FUNCTION_BLOCK FB_Robot EXTENDS FB_EquipmentModule_SR
VAR
    // Sub module definitions here

    // List of sub modules

    ipSubModules_Init : ARRAY[1..Parameters_PackML_Base.MAX_NO_OF_SUBMODULES] OF I_PackML_BaseModule := [];

    // Component definitions here

    Robot : FB_Component_Robot := (Name := 'Robot');

END_VAR

VAR

    //Properties
    DetailIndex : UDINT := 1;

    Handshake_Step : DINT;

    _DryRun : BOOL;

END_VAR

METHOD PROTECTED Aborting
VAR_INPUT
END_VAR
Handshake_Step                      := 0;
Robot.Handshake.OUT.Execute_Step    := FALSE;
Robot.Handshake.OUT.Execute_StepNum := 0;
DetailIndex                         := 1;

Super^.Aborting();
END_METHOD

METHOD PROTECTED Clearing
VAR_INPUT
END_VAR
Super^.Clearing();
END_METHOD

METHOD PROTECTED Completing
VAR_INPUT
END_VAR
Super^.Completing();
END_METHOD

METHOD CyclicLogic
VAR_INPUT
END_VAR

VAR

END_VAR
IF NOT _InitComplete THEN
    _InitComplete := Initialize();
    RETURN;
END_IF

//SimulationOn();

// transfer var from EM to COMP

// IF _Name = 'Robot 1' THEN

//     Robot.RobotType := 'Handling';

// ELSIF _Name = 'Robot 2' OR _Name = 'Robot 3' THEN

//     Robot.RobotType := 'Fastening';

// END_IF

SUPER^.CyclicLogic();
END_METHOD

METHOD CyclicLogicSimulation : BOOL
VAR_INPUT
END_VAR
END_METHOD

PROPERTY DryRun : BOOL
GET
DryRun := _DryRun;
END_GET
SET
_DryRun := DryRun;
END_SET
END_PROPERTY

METHOD PROTECTED Execute
VAR_INPUT
END_VAR
//  logic
WaitSync_Robot();

SubModuleMonitor();

SUPER^.Execute();
END_METHOD

METHOD ExtractNumFromString : DINT
VAR_INPUT
    InputString : STRING;
END_VAR

VAR
    NumberString : STRING     := ''; // Temporary string to collect digits
    Numbers      : STRING[10] := '0123456789'; // Temporary string to collect digits
    CurrentChar  : BYTE; // Current character being processed
    Result       : UDINT := 0; // Final extracted number as UDINT
    i            : INT   := 1; // String index
END_VAR
ExtractNumFromString := 0;
j                    := 0;

FOR i := 0 TO LEN(InputString) DO
    CurrentChar := InputString[i];

    // Check if the current character is a digit
    IF CurrentChar >= Numbers[0] AND CurrentChar <= Numbers[9] THEN
        NumberString[j] := CurrentChar;
        j               := j + 1;
    END_IF
END_FOR

// Check for a number at the end of the string
IF LEN(NumberString) > 0 THEN
    ExtractNumFromString := STRING_TO_DINT(NumberString); // Convert to UDINT
END_IF
END_METHOD

METHOD HMIControl
VAR_INPUT
END_VAR
END_METHOD

METHOD PROTECTED Holding
VAR_INPUT
END_VAR
IF Robot.Handshake.IN.TaskRunning = FALSE THEN
    SUPER^.Holding();
END_IF
END_METHOD

//! @summary Basic module initialization logic
METHOD PROTECTED Initialize : BOOL;
VAR
    i                        : UDINT;
    varInfo                  : __SYSTEM.VAR_INFO;
    AllSubUnitsInitialized   : BOOL := TRUE;
    AllComponentsInitialized : BOOL := TRUE;
END_VAR

//! @description This method is called by <c>CyclicLogic()</c> as required
Initialize := FALSE;

CASE DescendantSequenceState OF
    0:
        RegisterComponent(Robot);

        _LogModeChanges         := FALSE;
        _LogStateChanges        := FALSE;
        DescendantSequenceState := DescendantSequenceState + 10;

    10:
        //Setup Custom modes here

        (*CustomModes(eMode                          :=,
                    sName                          :=,
                    bDisableClearing               :=,
                    bDisableStarting               :=,
                    bDisableSuspended              :=,
                    bDisableStopping               :=,
                    bDisableAborting               :=,
                    bDisableHolding                :=,
                    bDisableHeld                   :=,
                    bDisableUnholding              :=,
                    bDisableSuspending             :=,
                    bDisableUnsuspending           :=,
                    bDisableResetting              :=,
                    bDisableIdle                   :=,
                    bDisableCompleting             :=,
                    bDisableComplete               :=,
                    bEnableUnitModeChangeStopped   :=,
                    bEnableUnitModeChangeIdle      :=,
                    bEnableUnitModeChangeSuspended :=,
                    bEnableUnitModeChangeExecute   :=,
                    bEnableUnitModeChangeAborted   :=,
                    bEnableUnitModeChangeHeld      :=,
                    bEnableUnitModeChangeComplete  :=,
                    bError                         =>,
                    nErrorId                       =>);*)

        DescendantSequenceState := DescendantSequenceState + 10;

    20:
        //Copy Mode names

        FOR i := 1 TO 3 DO
            ModeNames[i] := F_UnitModeToString(UDINT_TO_DINT(i));
        END_FOR

        RegisterExternalController(Controller := fbControlSourceHMI);
        fbControlSourceHMI.CyclicLogic();
        DescendantSequenceState := DescendantSequenceState + 10;

    30:
        //Call the Super

        IF SUPER^.Initialize() THEN
            DescendantSequenceState := DescendantSequenceState + 10;
        END_IF

    40:
        Initialize := TRUE;
END_CASE
END_METHOD

METHOD NailPlate : BOOL
VAR_INPUT
    Step : ST_CSV_Step;
END_VAR
// clear out array first
Robot.Clear_DataToSend();

// first entry is always step type
Robot.RecipeData_ToSend[1] := DINT_TO_USINT(E_CommandName.NailPlate);

// Robot.RecipeData_ToSend[2] := INT_TO_USINT(Plates[1].PlateNumber);
// 
// Robot.RecipeData_ToSend[3] := STRING_TO_USINT(Plates[1].PlateGauge);
// 
// Robot.RecipeData_ToSend[4] := LREAL_TO_USINT(TRUNC(Plates[1].PlateWidth * 10));
// 
// Robot.RecipeData_ToSend[5] := LREAL_TO_USINT(TRUNC(Plates[1].PlateHeight * 10));
// 
// Robot.RecipeData_ToSend[6] := LREAL_TO_USINT(TRUNC(Plates[1].PlatePlaceX * 10));
// 
// Robot.RecipeData_ToSend[7] := LREAL_TO_USINT(TRUNC(Plates[1].PlatePlaceY * 10));
// 
// Robot.RecipeData_ToSend[8] := LREAL_TO_USINT(TRUNC(Plates[1].PlatePlaceAngle * 10));
END_METHOD

PROPERTY OtherInputs : ARRAY[0..7] OF USINT
GET
OtherInputs := Robot.OtherInputs;
END_GET
END_PROPERTY

PROPERTY OtherOutputs : ARRAY[0..7] OF USINT
SET
Robot.OtherOutputs := OtherOutputs;
END_SET
END_PROPERTY

METHOD PROTECTED Resetting
VAR_INPUT
END_VAR
// reset handshake step
Handshake_Step                      := 0;
Robot.Handshake.OUT.Execute_Step    := FALSE;
Robot.Handshake.OUT.Execute_StepNum := 0;
DetailIndex                         := 1;

Super^.Resetting();
END_METHOD

METHOD PROTECTED Starting
VAR_INPUT
END_VAR
Handshake_Step                      := 0;
Robot.Handshake.OUT.Execute_Step    := FALSE;
Robot.Handshake.OUT.Execute_StepNum := 0;
DetailIndex                         := 1;

Super^.Starting();
END_METHOD

METHOD PROTECTED Stopping
VAR_INPUT
END_VAR
Super^.Stopping();
END_METHOD

(*! @summary This method monitors <b>submodules</b> within this PackML module and initiates fault responses as required*)
METHOD PROTECTED SubModuleMonitor : BOOL
SUPER^.SubModuleMonitor();
END_METHOD

METHOD PROTECTED Suspending
VAR_INPUT
END_VAR
IF Robot.Handshake.IN.TaskRunning = FALSE THEN
    SUPER^.Suspending();
END_IF
END_METHOD

METHOD PROTECTED Unholding
VAR_INPUT
END_VAR
SUPER^.Unholding();
END_METHOD

METHOD PROTECTED Unsuspending
VAR_INPUT
END_VAR
IF Robot.Handshake.IN.TaskRunning OR _InSimulation OR _ForceHold THEN
    SUPER^.Unsuspending();
END_IF
END_METHOD

METHOD WaitSync_Robot : BOOL
VAR
END_VAR

VAR_INST
    State : UDINT;
END_VAR
CASE State OF
    0:
        IF Robot.Handshake.IN.SubStepNumber > E_WaitSync.EMPTY THEN
            State := 1;
        END_IF

    1:
        _RequestedWaitSync := Robot.Handshake.IN.SubStepNumber;

        IF _RequestedWaitSync = _ResponseWaitSync THEN
            State := 2;
        END_IF

    2:
        Robot.Handshake.OUT.SubStepResponse := _ResponseWaitSync;

        IF Robot.Handshake.IN.SubStepNumber = E_WaitSync.EMPTY THEN
            _RequestedWaitSync := Robot.Handshake.IN.SubStepNumber;

            IF _ResponseWaitSync = E_WaitSync.EMPTY THEN
                Robot.Handshake.OUT.SubStepResponse := E_WaitSync.EMPTY;
                State                               := 0;
            END_IF
        END_IF

END_CASE
END_METHOD

END_FUNCTION_BLOCK

(* stored: Version 1.1.0.1
   POU FB_Robot: Id {1600db56-8704-42a5-b4ed-9569364dccae}, SpecialFunc None
   Folder I_CyclicFB: Id {f5633602-59b7-4bc0-9d4d-ad1c9ac3c89c}
   Folder Methods: Id {3c285524-643a-4343-a43c-a6df2c090b43}
   Folder ActingStates: Id {e4c87074-4e3f-4b79-aa36-c3b0b3bf226d}
   Folder CommandSteps: Id {61add708-9f29-4d83-adda-d2dcfb977e3f}
   Folder WaitingStates: Id {07ea4080-d9c0-4b39-9c64-a0a78873d1a8}
   Folder Properties: Id {e67c342a-5979-4627-bde3-a6f0dcd900b1}
   Method Aborting: Id {52fe1441-b0c0-423d-9d7a-ac2b065483cc}
   Method Clearing: Id {f68b84fa-c8c7-4a58-bb40-a12a77c808f3}
   Method Completing: Id {2b2dd47a-19b1-4d47-9ce0-79bec958c7ba}
   Method CyclicLogic: Id {86d8ffcb-cac6-4160-a90f-d2a7ddb84e46}
   Method CyclicLogicSimulation: Id {bb36d491-7e01-412f-8551-94b1c8ee0781}
   Property DryRun: Id {da5aa395-7e05-4bdc-a91b-eeaac04ecb7f}
   Get Get: Id {daac72f7-740e-4db6-a60b-9ab977f41f44}
   Set Set: Id {ecd88f42-46af-4430-82a5-7fa5e4ab3904}
   Method Execute: Id {18abe9ef-2c11-4fb0-bebc-eb0dad52c857}
   Method ExtractNumFromString: Id {96ae7f73-9467-4376-97ac-565ef616bc89}
   Method HMIControl: Id {28ac312f-fa82-4879-a674-1e946a88b00e}
   Method Holding: Id {b5937811-ff21-403d-b459-8391def9849f}
   Method Initialize: Id {33c7f9f5-feaf-4676-a2d5-65fc51e632d6}
   Method NailPlate: Id {f9b4837a-7316-49e5-92b5-e453cd7a3b8c}
   Property OtherInputs: Id {a2feda0e-e90f-4cdb-9a98-8d142025e152}
   Get Get: Id {572b02f7-6655-4d44-80d3-63a1e37224b6}
   Property OtherOutputs: Id {99596f22-c2b6-4278-88d3-85609ab5cea5}
   Set Set: Id {3263d4a6-5777-4a6d-bfd6-f347c43b4776}
   Method Resetting: Id {99efc620-e8f8-4a41-a023-b4a190f05cc0}
   Method Starting: Id {4000ad44-a0ea-48be-8105-bb74b62288e7}
   Method Stopping: Id {eb73f352-8881-4097-9d33-887f0f0cd3cb}
   Method SubModuleMonitor: Id {0f055ad8-7d39-4dd2-85e3-da4c2757804c}
   Method Suspending: Id {34e4640b-ef80-4f78-8429-8e25e6825505}
   Method Unholding: Id {2732c77c-cdba-42a7-9acd-90f892d1f837}
   Method Unsuspending: Id {1191d78b-8f90-4456-96f4-d6ad410ed060}
   Method WaitSync_Robot: Id {b1c430e7-ca0e-4ee7-8ade-43f3ebe7a29d} *)
